{attribute 'qualified_only'}
{attribute 'strict'}
TYPE E_Color :
(
	Red := 0,
	Blue := 1,
	Green:= 2
);
END_TYPE

(* stored: Version 1.1.0.1, ProductVersion 3.1.4024.16
   DUT E_Color: Id {4c8ff947-3fd4-4d5a-939a-b88059239d30} *)
